INTERFACE I_XtsNctBaseUnit

{attribute 'monitoring' := 'call'}
PROPERTY ActiveTime : REAL
GET
END_GET
END_PROPERTY

{attribute 'monitoring' := 'call'}
PROPERTY AnalogInput1 : LREAL
GET
END_GET
END_PROPERTY

{attribute 'monitoring' := 'call'}
PROPERTY AnalogInput2 : LREAL
GET
END_GET
END_PROPERTY

PROPERTY BIC : ARRAY[1..256] OF BYTE
GET
END_GET
SET
END_SET
END_PROPERTY

{attribute 'monitoring' := 'call'}
PROPERTY ControlVoltage : UINT
GET
END_GET
SET
END_SET
END_PROPERTY

{attribute 'monitoring' := 'call'}
PROPERTY DeviceName : STRING(31)
GET
END_GET
SET
END_SET
END_PROPERTY

{attribute 'monitoring' := 'call'}
PROPERTY DigitalInput1 : BOOL
GET
END_GET
END_PROPERTY

{attribute 'monitoring' := 'call'}
PROPERTY DigitalInput2 : BOOL
GET
END_GET
END_PROPERTY

{attribute 'monitoring' := 'call'}
PROPERTY DigitalInput3 : BOOL
GET
END_GET
END_PROPERTY

{attribute 'monitoring' := 'call'}
PROPERTY DigitalInput4 : BOOL
GET
END_GET
END_PROPERTY

{attribute 'monitoring' := 'call'}
PROPERTY DigitalOutput1 : BOOL
GET
END_GET
SET
END_SET
END_PROPERTY

{attribute 'monitoring' := 'call'}
PROPERTY DigitalOutput2 : BOOL
GET
END_GET
SET
END_SET
END_PROPERTY

{attribute 'monitoring' := 'call'}
PROPERTY DigitalOutput3 : BOOL
GET
END_GET
SET
END_SET
END_PROPERTY

{attribute 'monitoring' := 'call'}
PROPERTY DigitalOutput4 : BOOL
GET
END_GET
SET
END_SET
END_PROPERTY

{attribute 'monitoring' := 'call'}
PROPERTY HardwareVersion : STRING(3)
GET
END_GET
SET
END_SET
END_PROPERTY

{attribute 'monitoring' := 'call'}
PROPERTY Identity : REFERENCE TO ProductIdentity
GET
END_GET
SET
END_SET
END_PROPERTY

METHOD Initalize : REFERENCE TO ST_ReturnStructure

VAR_INPUT
	bExecute: BOOL;
END_VAR
END_METHOD

{attribute 'monitoring' := 'call'}
PROPERTY InputProcessData : REFERENCE TO ST_NctProcessData
GET
END_GET
END_PROPERTY

{attribute 'monitoring' := 'call'}
PROPERTY IsInterfaceAssigned : BOOL
GET
END_GET
END_PROPERTY

PROPERTY MoverGuid : GUID
GET
END_GET
SET
END_SET
END_PROPERTY

{attribute 'monitoring' := 'call'}
PROPERTY MoverUsername : STRING(31)
GET
END_GET
SET
END_SET
END_PROPERTY

PROPERTY NctBaseUnitInterface : I_TcIoXtsNctBaseUnitInterface
GET
END_GET
END_PROPERTY

{attribute 'monitoring' := 'call'}
PROPERTY OutputProcessData : REFERENCE TO ST_NctProcessData
GET
END_GET
SET
END_SET
END_PROPERTY

{attribute 'monitoring' := 'call'}
PROPERTY PwmChannel1 : LREAL
GET
END_GET
SET
END_SET
END_PROPERTY

{attribute 'monitoring' := 'call'}
PROPERTY PwmChannel2 : LREAL
GET
END_GET
SET
END_SET
END_PROPERTY

{attribute 'monitoring' := 'call'}
PROPERTY PwmChannel3 : LREAL
GET
END_GET
SET
END_SET
END_PROPERTY

{attribute 'monitoring' := 'call'}
PROPERTY PwmFrequency : LREAL
GET
END_GET
SET
END_SET
END_PROPERTY

METHOD ReadRegister : REFERENCE TO ST_ReturnStructure

VAR_INPUT
	bExecute		: BOOL;
	stRegisterType	: NctRegisterType;
END_VAR
END_METHOD

{attribute 'monitoring' := 'call'}
PROPERTY Status : REFERENCE TO NctBaseUnitStatus
GET
END_GET
END_PROPERTY

METHOD UpdateProcessData : REFERENCE TO ST_ReturnStructure

VAR_INPUT
	bEnable	: BOOL;	//Enables the cylcilc communication
END_VAR
END_METHOD

METHOD WriteRegister : REFERENCE TO ST_ReturnStructure

VAR_INPUT
	bExecute		: BOOL;
	stRegisterType	: NctRegisterType;
END_VAR
END_METHOD

END_INTERFACE

(* stored: Version 1.1.0.1, ProductVersion 3.1.4026.12
   Itf I_XtsNctBaseUnit: Id {2b310d87-b5c9-0572-3569-3110c4511371}
   Folder Methods: Id {63d72e80-4ea2-009a-3541-66552460be54}
   Folder Adminstrative: Id {9205234a-5316-0dca-0a23-68e3a1bab8df}
   Folder Communication: Id {45a9adb1-128d-0a6f-0bde-ffe00d1b4231}
   Folder Properties: Id {40dfb317-344c-0b4d-20fd-63c2ce39487c}
   Folder Administrative: Id {4f73fc20-5c93-0217-05ff-f0d05fcbc58f}
   Folder ProcessData: Id {06b94ea2-390b-03da-0be2-7bd9a6699615}
   Folder ProcessImage: Id {46713149-e4cd-0871-0114-b2b46929c886}
   Folder Registers: Id {c1594288-4628-0bb2-27f5-268e0e0c1b08}
   Property ActiveTime: Id {71e6e6b6-4cfa-0c37-2665-24b2d4f6e385}
   Get Get: Id {fd6f318e-9647-0cfb-2b06-7c2ec8fe49ff}
   Property AnalogInput1: Id {adc2595b-ce98-0239-1a79-d1ff88832e95}
   Get Get: Id {59e41706-22dd-068d-0c15-318790bfff85}
   Property AnalogInput2: Id {64e7a36d-8885-08fa-370b-9f047f45a15f}
   Get Get: Id {43c0b538-1c91-0579-2991-7dbead668437}
   Property BIC: Id {939e10f2-36f7-0421-355f-c518e6d6a2f8}
   Get Get: Id {b7c5e17d-e9cb-0fea-0f5b-81597832d71d}
   Set Set: Id {08f4b4ed-da11-02ea-0d43-33fcc20a37c1}
   Property ControlVoltage: Id {dd61dbc8-706d-0d65-16d0-16d25d639d14}
   Get Get: Id {01050729-c3b9-0371-0238-d07078aa5955}
   Set Set: Id {a15526a9-be53-069c-19fa-222902eb1f5e}
   Property DeviceName: Id {73926f5c-717f-040c-0b53-0a39046aae6d}
   Get Get: Id {545dfc1d-2fb2-0ce6-2da5-36a6d90c3065}
   Set Set: Id {0a8f9bcc-d158-0f17-359b-fe2b575c8409}
   Property DigitalInput1: Id {3390b9f3-5cee-0006-2c02-b82b947c5fdb}
   Get Get: Id {8dfe1a88-0707-0192-2346-08e62b75a65e}
   Property DigitalInput2: Id {1ee2d02e-8cf1-0eae-3a56-ebb02e9b148c}
   Get Get: Id {7ff759d5-d4b7-0464-1af5-6548a4d916f5}
   Property DigitalInput3: Id {6f309c75-e863-063b-3a63-eaa666e80cbb}
   Get Get: Id {29f00595-abd2-09e7-2202-b852c88a56c4}
   Property DigitalInput4: Id {2d35c20e-24e6-0396-0474-a30310b42469}
   Get Get: Id {61bfd6b2-9949-0570-2a62-fd020e2eb615}
   Property DigitalOutput1: Id {94fc6155-cad9-019e-3d3a-d34938920530}
   Get Get: Id {68fca6e9-36cf-08bd-1578-0c662148b4e9}
   Set Set: Id {abafc4f0-471d-0d8a-37ae-8fcdb726809c}
   Property DigitalOutput2: Id {34fc016d-ddf4-0b1b-134e-784fc5c26c47}
   Get Get: Id {b2c796f1-8ab6-0bb5-1994-a5f045e32a42}
   Set Set: Id {13f87e64-ac85-05b7-1a42-9c4528cca52f}
   Property DigitalOutput3: Id {9e129d78-aa10-0a2c-0bc0-b3fc461bdd20}
   Get Get: Id {d91165d2-2ec5-0342-1104-dcd6b5180e0a}
   Set Set: Id {10f67b76-db64-0983-0cea-b3fe158ede37}
   Property DigitalOutput4: Id {a1c5830d-d51d-08d9-2fe9-0fd6f1cae003}
   Get Get: Id {f3ab0b38-f2f0-042b-2005-a588ce925f4b}
   Set Set: Id {2d3faead-e594-0172-0b2e-046b787fecce}
   Property HardwareVersion: Id {9eea95aa-4a18-05e4-1ab9-380bf78598e9}
   Get Get: Id {7fc0792b-e2ec-0472-12a3-46df27b3e18b}
   Set Set: Id {28655299-0017-0d1b-1ccb-8887303f60fa}
   Property Identity: Id {60c4c51e-3aca-0b8c-0418-a83bd3bb6bf2}
   Get Get: Id {21f3663d-7085-0182-2f44-d79c8eb958e4}
   Set Set: Id {d530708d-3577-00cc-0b34-d205d2f30295}
   Method Initalize: Id {ac939d7e-388d-0f75-2bce-48cf494eedb2}
   Property InputProcessData: Id {ea514186-a31f-0586-2957-378f30a9838a}
   Get Get: Id {b43059a2-430d-04ea-12f7-2cedecf652e7}
   Property IsInterfaceAssigned: Id {6adcdacc-e473-01ca-3529-2326a002af16}
   Get Get: Id {c9cb23f1-e348-0f4a-1f05-fc11b4e39503}
   Property MoverGuid: Id {677a5f94-ce88-0061-3fd9-0705452d511f}
   Get Get: Id {550eb63d-4ed0-04bc-2a7b-0f7031b97cc8}
   Set Set: Id {d0e36f74-f189-034a-2a28-ad7f6f8c9e4a}
   Property MoverUsername: Id {2f2b38db-c0fd-0aea-1aae-154c85925606}
   Get Get: Id {b7c3b576-16f1-017a-2065-3cb1fb1e0c07}
   Set Set: Id {a4dbef06-a3c1-0994-1a8f-53e8b045e452}
   Property NctBaseUnitInterface: Id {350e3b2f-a26b-0c01-0c45-402c0a46f1dd}
   Get Get: Id {5a62bd65-7b16-0acb-1841-fb72ab5afa4a}
   Property OutputProcessData: Id {68b5b51f-4300-07e8-392a-21c8a56b3bfc}
   Get Get: Id {b10b8511-10b7-022a-3e20-13ba02471480}
   Set Set: Id {65a94411-a0fb-07be-0b52-66d0a4766baf}
   Property PwmChannel1: Id {30ded0ac-cc1d-00ea-28cc-6f23182de97e}
   Get Get: Id {32012a30-5559-0dfa-2266-2874aa2de1e7}
   Set Set: Id {89f1318c-175d-0016-192b-e802f332bc89}
   Property PwmChannel2: Id {869eb77d-0535-04f3-2536-d0a85bd4795a}
   Get Get: Id {5ad31de3-5cd6-0e0c-28fa-05a116fc94b0}
   Set Set: Id {a481c708-c11e-0ef2-37a5-357eb312b458}
   Property PwmChannel3: Id {1f00b17e-6715-0235-01f0-dbcfa3803208}
   Get Get: Id {d402e35e-7db6-0da2-1707-80258b511640}
   Set Set: Id {ac36fa5a-2999-0172-240f-0daa3cfcb0db}
   Property PwmFrequency: Id {4a603542-fec6-005b-1e16-989bf6084089}
   Get Get: Id {8dc85e96-8f4b-0d29-23a4-39535415458c}
   Set Set: Id {1fc69d12-7416-0be3-30e4-49734ff65f7d}
   Method ReadRegister: Id {bea69afb-468e-0cdb-08ae-32fc9e78e5fa}
   Property Status: Id {450b05c8-a1ba-070b-00f7-f15b1ec9a635}
   Get Get: Id {bdbfefe4-1739-0b3b-015a-d84a5bedc31f}
   Method UpdateProcessData: Id {716f09e6-de9d-0823-2042-ba588278d67c}
   Method WriteRegister: Id {fe33a921-a0a3-09f2-05b3-63b915a0687e} *)
